FUNCTION_BLOCK FB_Triamec
VAR_INPUT
END_VAR
VAR_OUTPUT
END_VAR
VAR
END_VAR

END_FUNCTION_BLOCK

(* stored: Version 1.1.0.1, ProductVersion 3.1.4024.12
   POU FB_Triamec: Id {23682737-03b6-4da5-afce-708bad80b677}, SpecialFunc None *)
